# EPICS substitutions: oerconeSup/unit_setter.substitutions
file $(UTILITIES)/db/unit_setter.template {
  pattern
    {P,    FROM, TO}

    {"\$(P)", "UNITS", "PRESSURE"}
}
